{attribute 'strict'}
TYPE E_CognexCameraGetValuesState :
(
	CAMERA_GET_VALUES_SEND_COMMAND_VALUE_1		:= 0,
	CAMERA_GET_VALUES_RECEIVE_RESPONSE_VALUE_1	:= 10,
	CAMERA_GET_VALUES_SEND_COMMAND_VALUE_2		:= 20,
	CAMERA_GET_VALUES_RECEIVE_RESPONSE_VALUE_2	:= 30,
	CAMERA_GET_VALUES_SEND_COMMAND_VALUE_3		:= 40,
	CAMERA_GET_VALUES_RECEIVE_RESPONSE_VALUE_3	:= 50,
	CAMERA_GET_VALUES_SEND_COMMAND_VALUE_4		:= 60,
	CAMERA_GET_VALUES_RECEIVE_RESPONSE_VALUE_4	:= 70,
	CAMERA_GET_VALUES_GETTING_DONE				:= 80
);
END_TYPE

(* stored: Version 1.1.0.1, ProductVersion 3.1.4024.12
   DUT E_CognexCameraGetValuesState: Id {a2e7b000-5043-43c4-a1fa-1f4116f07773} *)
